// TwinCAT 3 PLC project CheckerFunctions
// ProgramVersion: 3.1.4024.0
// libraries:
//   Tc2_Standard, * (Beckhoff Automation GmbH)
//   Tc2_System, * (Beckhoff Automation GmbH)
//   Tc3_Module, * (Beckhoff Automation GmbH)
// project tree:
//   / PlcTask.TcTTO
//   POUs/ CheckBounds.TcPOU, CheckDivByte.TcPOU, CheckDivReal.TcPOU, CheckDivWord.TcPOU, CheckRangeInt.TcPOU, CheckRangeSigned.TcPOU, MAIN.TcPOU
// real-time tasks:
//   TASK PlcTask: cycle T#10ms, priority 20, ADS port 350
//   TASK PlcTask1: cycle T#10ms, priority 21, ADS port 351
//   TASK PlcTask2: cycle T#10ms, priority 22, ADS port 352
//   TASK PlcTask3: cycle T#10ms, priority 23, ADS port 353
//   TASK PlcTask4: cycle T#10ms, priority 24, ADS port 354
//   TASK PlcTask5: cycle T#10ms, priority 25, ADS port 355
//   TASK PlcTask6: cycle T#10ms, priority 26, ADS port 356
//   TASK PlcTask7: cycle T#10ms, priority 27, ADS port 357

CONFIGURATION CheckerFunctions
    RESOURCE PLC ON TwinCAT3
        TASK PlcTask(INTERVAL := T#10ms, PRIORITY := 20);
        PROGRAM MAIN WITH PlcTask : MAIN;
    END_RESOURCE
END_CONFIGURATION

// ---- POUs/MAIN.TcPOU
PROGRAM MAIN
VAR
// 1. CheckBounds aan die de waarde tussen 15 en 24 regelt
waarde : DINT;       // De waarde die je wilt controleren
gecorrigeerdeWaarde : DINT;

// 2. CheckDivByte
testDivisor : BYTE;
result : BYTE;

// 3. CheckDivReal? Int staat niet op infosys
erg : REAL; // Resultaat van de deling
v1 : REAL := 799; // De dividend
d : REAL; // De divisor

// 4. CheckDivWord
resultREAL : REAL;
dividend : WORD := 1000; // Vervang door de waarde die je wilt delen
divisor : WORD := 0;     // Vervang door de waarde waardoor je wilt delen

// 5. CheckRangeSigned
getesteWaarde : DINT;
resultaat : DINT;
minGrens : DINT := -4095; // Definieer de ondergrens van het bereik
maxGrens : DINT := 4095;  // Definieer de bovengrens van het bereik

// 6. CheckRangeInt met TYPES voor waarden van 0 t.e.m. 32.767
testValue : INT; // De waarde die je wilt testen
checkedValue : INT;

END_VAR

// Checker functions
// Maak de checker functions aan die gezien werden tijdens de les:

// 1. CheckBounds aan die de waarde tussen 15 en 24 regelt
waarde := 26; // Een voorbeeldwaarde
gecorrigeerdeWaarde := CheckBounds(waarde, 15, 24);

// 2. CheckDivByte
testDivisor := 0; // Test met een divisor van 0
result := CheckDivByte(testDivisor);

// 3. CheckDivReal? Int staat niet op infosys
d := 0; // Stel de divisor in op een waarde die getest moet worden, bijvoorbeeld 0
d := CheckDivReal(d); // Roep de CheckDivReal functie aan om te controleren op deling door nul

erg := v1 / d; // Voer de deling uit met de gecontroleerde divisor

// 4. CheckDivWord
divisor := CheckDivWord(divisor); // Controleer de divisor
resultREAL := WORD_TO_REAL(dividend) / WORD_TO_REAL(divisor); // Voer de deling uit

// 5. CheckRangeSigned
// Stel de te testen waarde in
getesteWaarde := 5000; // Een waarde buiten het bereik om de functionaliteit te testen

// Roep de CheckRangeSigned functie aan om de waarde te controleren en aan te passen
resultaat := CheckRangeSigned(getesteWaarde, minGrens, maxGrens);

// 6. CheckRangeInt met TYPES voor waarden van 0 t.e.m. 32.767
// Test de functie met een waarde buiten het bereik
testValue := 40000; // Een waarde boven het maximale bereik
checkedValue := CheckRangeInt(testValue); // Zou 32767 moeten retourneren

END_PROGRAM

// ---- POUs/CheckBounds.TcPOU
FUNCTION CheckBounds : DINT
VAR_INPUT
    i, l, u : DINT;
END_VAR

IF i<l THEN
    CheckBounds := l;
ELSIF i>u THEN
    CheckBounds := u;
ELSE
    CheckBounds := i;
END_IF

END_FUNCTION

// ---- POUs/CheckDivByte.TcPOU
FUNCTION CheckDivByte : BYTE
VAR_INPUT
    divisor : BYTE;
END_VAR
VAR
END_VAR

IF divisor = 0 THEN
    CheckDivByte := 1;(**)
ELSE
    CheckDivByte := divisor;
END_IF

END_FUNCTION

// ---- POUs/CheckDivReal.TcPOU
FUNCTION CheckDivReal : REAL
VAR_INPUT
    divisor : REAL;
END_VAR
VAR
END_VAR

IF divisor = 0 THEN
    CheckDivReal := 1;
ELSE
    CheckDivReal := divisor;
END_IF

END_FUNCTION

// ---- POUs/CheckDivWord.TcPOU
FUNCTION CheckDivWord : WORD
VAR_INPUT
    divisor : WORD;
END_VAR
VAR
END_VAR

IF divisor = 0 THEN
    CheckDivWord := 1;
ELSE
    CheckDivWord := divisor;
END_IF

END_FUNCTION

// ---- POUs/CheckRangeSigned.TcPOU
FUNCTION CheckRangeSigned : DINT
VAR_INPUT
    value, lower, upper: DINT;
END_VAR

IF (value < lower) THEN
    CheckRangeSigned := lower;
ELSIF(value > upper) THEN
    CheckRangeSigned := upper;
ELSE
    CheckRangeSigned := value;
END_IF

END_FUNCTION

// ---- POUs/CheckRangeInt.TcPOU
FUNCTION CheckRangeInt : INT
VAR_INPUT
    valueint : INT;
END_VAR

VAR CONSTANT
lowerBound : INT := 0;
upperBound : INT := 32767;
END_VAR

// Controleer of de waarde binnen het bereik ligt en corrigeer deze indien nodig
IF valueint < lowerBound THEN
    CheckRangeInt := lowerBound;
ELSIF valueint > upperBound THEN
    CheckRangeInt := upperBound;
ELSE
    CheckRangeInt := valueint;
END_IF

END_FUNCTION
